(* IEC 61131-3 sources: cybercode_codesys_lib/src/communication, 5 files *)

(* ---- U_ByteToWord.st ---- *)
TYPE U_ByteToWord :
UNION
	wTag: WORD;
	bTag: ARRAY [0..1] OF BYTE;
END_UNION
END_TYPE

(* ---- U_RealToWord.st ---- *)
TYPE U_RealToWord :
UNION
	wTag: ARRAY [0..1] OF WORD;
	rTag: REAL;
END_UNION
END_TYPE

(* ---- FC_SwapBytesInWord .st ---- *)
FUNCTION FC_SwapBytesInWord : WORD
VAR_INPUT
    wInputValue : WORD;                     // Входное значение WORD
END_VAR
VAR
    uByteConverter : U_ByteToWord;          // Конвертер для работы с байтами
END_VAR

// Загружаем входное значение в конвертер
uByteConverter.wTag := wInputValue;

// Меняем местами байты: младший байт становится старшим, старший - младшим
FC_SwapBytesInWord := SHL(TO_WORD(uByteConverter.bTag[0]), 8) OR TO_WORD(uByteConverter.bTag[1]);

END_FUNCTION

(* ---- FC_SwapBytesInWordArray .st ---- *)
FUNCTION FC_SwapBytesInWordArray : ARRAY [0..1] OF WORD
VAR_INPUT
    awInputArray : ARRAY [0..1] OF WORD;    // Входной массив из двух WORD
END_VAR
VAR
    uByteConverter : U_ByteToWord;           // Конвертер для работы с байтами
    awOutputArray : ARRAY [0..1] OF WORD;   // Выходной массив
END_VAR

// Обработка первого WORD (индекс 0)
uByteConverter.wTag := awInputArray[0];
// Меняем местами байты и записываем в выходной массив
awOutputArray[0] := SHL(TO_WORD(uByteConverter.bTag[0]), 8) OR TO_WORD(uByteConverter.bTag[1]);

// Обработка второго WORD (индекс 1)
uByteConverter.wTag := awInputArray[1];
// Меняем местами байты и записываем в выходной массив
awOutputArray[1] := SHL(TO_WORD(uByteConverter.bTag[0]), 8) OR TO_WORD(uByteConverter.bTag[1]);

// Возвращаем преобразованный массив
FC_SwapBytesInWordArray := awOutputArray;

END_FUNCTION

(* ---- FC_SwapWordArrayElements .st ---- *)
FUNCTION FC_SwapWordArrayElements : ARRAY [0..1] OF WORD
VAR_INPUT
    awInputArray : ARRAY [0..1] OF WORD;    // Входной массив из двух WORD
END_VAR
VAR
    awOutputArray : ARRAY [0..1] OF WORD;   // Выходной массив
END_VAR

// Меняем местами элементы массива: [0] -> [1], [1] -> [0]
awOutputArray[0] := awInputArray[1];
awOutputArray[1] := awInputArray[0];

// Возвращаем массив с переставленными элементами
FC_SwapWordArrayElements := awOutputArray;

END_FUNCTION
